PROGRAM MAIN


VAR
	stRawIn		:	ST_CSL_RawIn;
	stRawOut	:	ST_CSL_RawOut;
	stIn		:	ST_CSL_In;
	stOut		: 	ST_CSL_Out;
	stParams	:	ST_CSL_Params; 
	
	estep 	: E_Step;
	
	
	timer	: TON();
	fb	: FB_MSF_Pistoni;
	
	slots	: INT;
	iMotors	: INT	:= 0;
	
	nerrid	: DINT; 
	
END_VAR

stRawout.bMotor	:= TRUE;
IF stRawin.bPieceSensorOutput THEN
	stRawout.bMotor	:= FALSE;
	timer (IN:= (stRawin.bPieceSensorOutput), PT := T#1000MS);
		IF timer.Q	THEN
		fb(
	bEnable:= NOT(stIn.bEmerg), 
	slot:= slots, 
	iMotor:= iMotors, 
	st_In:= stIn, 
	st_Params:= stParams, 
	st_Out:= stOut, 
	eStep=>  estep, 
	eErrStep=> estep, 
	nErrid=> nerrid);
		END_IF
END_IF

END_PROGRAM

(* stored: Version 1.1.0.1, ProductVersion 3.1.4024.12
   POU MAIN: Id {63e7df63-7f3f-44d1-9324-af642dc6ce72}, SpecialFunc None *)
